(* PLC project illuminated_button, Dassault Systèmes ControlBuild 2024x *)
(* stored: creationDateTime 2023-10-03T11:13:22-01:00 *)

(* This module simulates an illuminated push button with a momentary contact. *)
FUNCTION_BLOCK equipment_library.illuminated_button
  VAR_INPUT
    luminous : BOOL := false;
  END_VAR
  VAR_OUTPUT
    PB : BOOL := false;
  END_VAR
  VAR
    timeCounter : REAL := 0.0;
    action : BOOL := false;
  END_VAR
  VAR CONSTANT
    pulseDuration : REAL := 5.0;
    PBLogic : BOOL := true;
  END_VAR

(* -----------------------------------------------------------------	*)
(* Type : Model of Operative Behaviour					*)
(* Category :  Power								*)
(* Author : Dassault Systemes						*)
(* Update date : June 2018							*)
(* -----------------------------------------------------------------	*)
(* This module simulates an illuminated push button			*)
(* with a momentary contact.						*)
(* -----------------------------------------------------------------	*)

IF (action) THEN
	timeCounter := timeCounter + ( CLOCK_PERIOD / 1000000.0);
	IF (timeCounter > pulseDuration) THEN
		action := FALSE;
		timeCounter := 0.0;
	END_IF;
END_IF;
PB := (action XOR NOT PBLogic);
END_FUNCTION_BLOCK
